FUNCTION_BLOCK fb_IBN_Ventil_ohne_Log
VAR_INPUT
	AUTO_AUF : BOOL;
	VERFAHRZEIT : TIME;
END_VAR
VAR_OUTPUT
	RM_AUF : BOOL;
	RM_ZU  : BOOL;
END_VAR
VAR
	TON_AUF : Tc2_Standard.TON;
	TON_ZU 	: Tc2_Standard.TON;
END_VAR

	
IF AUTO_AUF THEN
	//Rückmeldung 	
	RM_ZU := FALSE;	
	TON_ZU(IN := FALSE);
	
	TON_AUF(IN := NOT RM_ZU, PT := VERFAHRZEIT);	
	RM_AUF := TON_AUF.Q ;	
ELSE
	//Rückmeldung 	
	RM_AUF := FALSE;	
	TON_AUF(IN := FALSE);
	
	TON_ZU(IN := NOT RM_AUF, PT := VERFAHRZEIT);
	RM_ZU := TON_ZU.Q ;	

END_IF

END_FUNCTION_BLOCK

(* stored: Version 1.1.0.1, ProductVersion 3.1.4024.11
   POU fb_IBN_Ventil_ohne_Log: Id {cbfde30d-efdb-448c-98af-bfca885d64cd}, SpecialFunc None *)
